INTERFACE I_PackML_IdleCommands

METHOD PUBLIC Abort
VAR_INPUT
END_VAR
END_METHOD

METHOD PUBLIC Start
VAR_INPUT
END_VAR
END_METHOD

METHOD PUBLIC Stop
VAR_INPUT
END_VAR
END_METHOD

END_INTERFACE

(* stored: Version 1.1.0.1, ProductVersion 3.1.4024.12
   Itf I_PackML_IdleCommands: Id {98a18d41-1301-03fd-1f24-fccf520ed562}
   Method Abort: Id {d6dbb4a1-b362-03fb-14fc-0a6c8d4ad1ee}
   Method Start: Id {10ff5ee6-413f-0d0d-317f-29627efddc1f}
   Method Stop: Id {430f4343-8497-0a2b-06a6-5e966e7fdc66} *)
